TEXTLIST LoadPriority
  0 = 'LoadPriority_None'
  1 = 'LoadPriority_Line0'
  2 = 'LoadPriority_Line1'
   = ''
END_TEXTLIST

(* stored: Version 1.1.0.1, ProductVersion 3.1.4024.3
   TextList LoadPriority: Id {911df754-24ad-49d2-bb51-70c059bbd455} *)
